FUNCTION_BLOCK FB_MultiActuator_NoFeedback
VAR_GENERIC CONSTANT
	LenActuators : UDINT := 1;
END_VAR
VAR
	Actuator : ARRAY[0..LenActuators-1] OF FB_Actuator_NoFeedback;
END_VAR

END_FUNCTION_BLOCK

(* stored: Version 1.1.0.1
   POU FB_MultiActuator_NoFeedback: Id {d05c1bbd-636f-44b6-915c-efafb64a4c0d}, SpecialFunc None *)
